(* generates a square wave with user-defined period and 50% duty cycle, min PLC task time = 100us *)
FUNCTION_BLOCK FB_SquareWave
VAR_INPUT
	bEnable			: BOOL;		(* set TRUE to enable pulse generation *)
	tPeriod			: TIME;		(* base period for pulse output, max period = T#4d *)
END_VAR
VAR_OUTPUT
	bOutput			: BOOL;		(* square wave output *)
	bRisingEdge		: BOOL;		(* TRUE = rising edge of bOutput *)
	bFallingEdge	: BOOL;		(* TRUE = falling edge of bOutput *)
END_VAR
VAR
	fbPulseTrain	: FB_PulseTrain;
END_VAR
(*
-------------------------------------------------------------------------------------------------
Date		Version	Author	Comments
-------------------------------------------------------------------------------------------------
30/01/2015	3.00.00	PB		No change

-------------------------------------------------------------------------------------------------
05/02/2010	1.00.00	PB		Initial release

-------------------------------------------------------------------------------------------------
*)

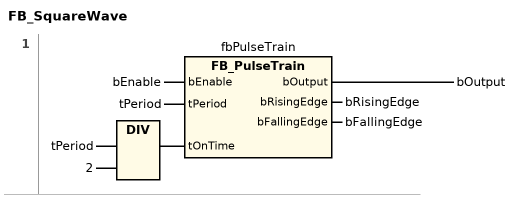
// NETWORK 1
fbPulseTrain(
    bEnable := bEnable,
    tPeriod := tPeriod,
    tOnTime := tPeriod / 2,
    bRisingEdge => bRisingEdge,
    bFallingEdge => bFallingEdge); // FB_PulseTrain
bOutput := fbPulseTrain.bOutput;

END_FUNCTION_BLOCK

(* stored: Version 1.1.0.1, ProductVersion 3.1.4024.15
   POU FB_SquareWave: Id {0ad12106-f1b5-4660-add7-a3b006335c94}, SpecialFunc None *)
